// TIA Portal project "Projeto Automação Industrial" (V15.1)
// Vorlageprojekt für das Buch mit Zielsystem S7-1200

(* hardware
DEVICE "S7-1200-Station_1"  S7-1200 Station
   slot 0: "Baugruppenträger_0"  Rack  V1.0
   slot 1: "PLC_1"  CPU 1211C DC/DC/DC  6ES7 211-1AE40-0XB0  V4.1
*)

// ===== PLC "PLC_1"  CPU 1211C DC/DC/DC =====

VAR_GLOBAL   // PLC tag table "Standard-Variablentabelle"
   "Conveyor1" AT %A0.0 : Bool;
   "At exit" AT %E0.0 : Bool;
   "Start" AT %E0.1 : Bool;
   "Start light" AT %Q1.1 : Bool;
   "Start_All" AT %Q3.0 : Bool;
   "Sorter 1" AT %Q2.1 : Bool;
   "Sorter 2" AT %Q2.2 : Bool;
   "Sorter 3" AT %Q2.3 : Bool;
   "Stop blade" AT %Q0.1 : Bool;
   "Sorter 1 turn" AT %Q0.3 : Bool;
   "Sorter 1 belt" AT %Q0.4 : Bool;
   "Stop conveyor" AT %Q2.4 : Bool;
   "Vision Sensor" AT %ID30 : DInt;
   "Counter 1" AT %QD30 : DInt;
   "Stop" AT %I0.3 : Bool;
   "Counter 1 exit" AT %Q2.5 : Bool;
   "Start/stop conveyor timer" AT %Q2.6 : Bool;
   "Counter 2" AT %QD34 : DInt;
   "Counter 2 exit" AT %Q2.7 : Bool;
   "Counter 3" AT %QD38 : DInt;
   "Counter 3 exit" AT %Q1.4 : Bool;
   "Conveyor2" AT %Q0.2 : Bool;
   "Sorter 2 turn" AT %Q0.5 : Bool;
   "Sorter 2 belt" AT %Q0.6 : Bool;
   "Sorter 3 turn" AT %Q0.7 : Bool;
   "Sorter 3 belt" AT %Q1.0 : Bool;
   "Stop Light" AT %Q1.3 : Bool;
   "Exited" AT %Q3.1 : Bool;
   "Exit Timer" AT %Q3.2 : Bool;
   "Reset" AT %I0.2 : Bool;
   "Reset Light" AT %Q1.2 : Bool;
END_VAR

// folder: System blocks/Program resources

DATA_BLOCK "IEC_Counter_0_DB"   // DB1
{ S7_Optimized_Access := 'TRUE' }
AUTHOR : Simatic
FAMILY : IEC
NAME : CNTR
VERSION : 1.0
// stored: InstanceOfName IEC_COUNTER
"IEC_COUNTER"
BEGIN
END_DATA_BLOCK

DATA_BLOCK "IEC_Timer_0_DB"   // DB2
{ S7_Optimized_Access := 'TRUE' }
AUTHOR : Simatic
FAMILY : IEC
NAME : IEC_TMR
VERSION : 1.0
// stored: InstanceOfName IEC_TIMER
"IEC_TIMER"
BEGIN
END_DATA_BLOCK

DATA_BLOCK "IEC_Timer_0_DB_4"   // DB3
{ S7_Optimized_Access := 'TRUE' }
AUTHOR : Simatic
FAMILY : IEC
NAME : IEC_TMR
VERSION : 1.0
// stored: InstanceOfName IEC_TIMER
"IEC_TIMER"
BEGIN
END_DATA_BLOCK

DATA_BLOCK "IEC_Counter_0_DB_1"   // DB5
{ S7_Optimized_Access := 'TRUE' }
AUTHOR : Simatic
FAMILY : IEC
NAME : CNTR
VERSION : 1.0
// stored: InstanceOfName IEC_COUNTER
"IEC_COUNTER"
BEGIN
END_DATA_BLOCK

DATA_BLOCK "IEC_Counter_0_DB_2"   // DB6
{ S7_Optimized_Access := 'TRUE' }
AUTHOR : Simatic
FAMILY : IEC
NAME : CNTR
VERSION : 1.0
// stored: InstanceOfName IEC_COUNTER
"IEC_COUNTER"
BEGIN
END_DATA_BLOCK

DATA_BLOCK "IEC_Timer_0_DB_2"   // DB7
{ S7_Optimized_Access := 'TRUE' }
AUTHOR : Simatic
FAMILY : IEC
NAME : IEC_TMR
VERSION : 1.0
// stored: InstanceOfName IEC_TIMER
"IEC_TIMER"
BEGIN
END_DATA_BLOCK

DATA_BLOCK "IEC_Timer_0_DB_1"   // DB8
{ S7_Optimized_Access := 'TRUE' }
AUTHOR : Simatic
FAMILY : IEC
NAME : IEC_TMR
VERSION : 1.0
// stored: InstanceOfName IEC_TIMER
"IEC_TIMER"
BEGIN
END_DATA_BLOCK

DATA_BLOCK "IEC_Timer_0_DB_3"   // DB9
{ S7_Optimized_Access := 'TRUE' }
AUTHOR : Simatic
FAMILY : IEC
NAME : IEC_TMR
VERSION : 1.0
// stored: InstanceOfName IEC_TIMER
"IEC_TIMER"
BEGIN
END_DATA_BLOCK

// folder: (top level)

FUNCTION "MHJ-PLC-Lab-Function-S71200" : Void   // FC9000, SCL
{ S7_Optimized_Access := 'TRUE' }
VERSION : 0.1
   VAR_TEMP
      rdTimeReturn : Int;
      outputTime : DTL;
      SyncVal : Byte;
      forVal : Int;
      forVal_2 : Int;
      Value : Byte;
   END_VAR
   VAR CONSTANT
      CompVal : Byte := 16#34;
      Value_01 : Byte := 16#11;
      Value_01_DW : DWord := 16#A165_D992;
      Value_02_DW : DWord := 16#58BE_4401;
   END_VAR
BEGIN

   #Value:=PEEK(area := 16#82,
        dbNumber := 0,
        byteOffset := 511);
   #Value := #Value + 1;

   POKE(area := 16#82,
        dbNumber := 0,
        byteOffset := 511,
        value := #Value);

   POKE(area:=16#81,
        dbNumber:=0,
        byteOffset:=1016,
        value:=#Value_01_DW);
   POKE(area := 16#81,
        dbNumber := 0,
        byteOffset := 1020,
        value := #Value_02_DW);

   POKE(area := 16#81,
        dbNumber := 0,
        byteOffset := 511,
        value := B#16#00);

   FOR #forVal := 0 TO 120 DO
       FOR #forVal_2:=0 TO 10 DO
           #rdTimeReturn:=RD_SYS_T(#outputTime);
           #rdTimeReturn := WR_SYS_T(#outputTime);
           #rdTimeReturn := RD_SYS_T(#outputTime);
           #rdTimeReturn := WR_SYS_T(#outputTime);
       END_FOR;
       #SyncVal:= PEEK(area := 16#81,
                      dbNumber := 0,
                      byteOffset := 511);
       IF #SyncVal = #CompVal THEN
          GOTO M_1;
       END_IF;
   END_FOR;
   RETURN;

   M_1:
   POKE(area := 16#81,
        dbNumber := 0,
        byteOffset := 511,
        value := B#16#0);
END_FUNCTION

ORGANIZATION_BLOCK "Main"   // OB1, LAD, ProgramCycle
TITLE = "Main Program Sweep (Cycle)"
{ S7_Optimized_Access := 'TRUE' }
VERSION : 0.1
   VAR_INPUT
      Initial_Call : Bool;   // Initial call of this OB
      Remanence : Bool;   // =True, if remanent data are available
   END_VAR
BEGIN

REGION Network 1
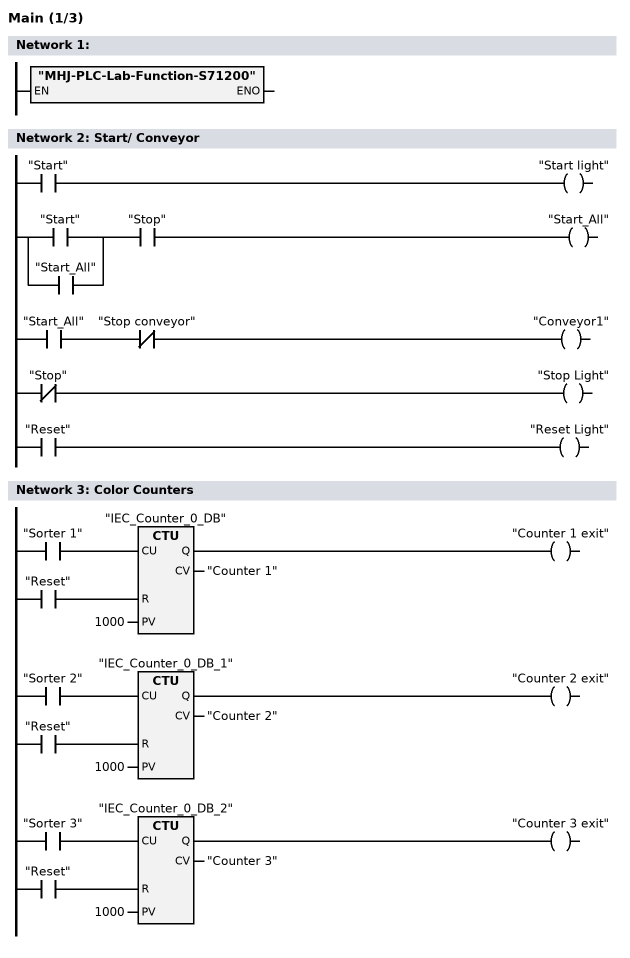
   RUNG wire#powerrail
      "MHJ-PLC-Lab-Function-S71200"()
   END_RUNG
   // the same network as SCL:
   "MHJ-PLC-Lab-Function-S71200"();
END_REGION

REGION Network 2: Start/ Conveyor
   RUNG wire#powerrail
      Contact( "Start" )
      Coil( "Start light" )
   END_RUNG
   RUNG wire#powerrail
      Contact( "Start" )
      wire#w1
      Contact( "Stop" )
      Coil( "Start_All" )
   END_RUNG
   RUNG wire#powerrail
      Contact( "Start_All" )
   END_RUNG wire#w1
   RUNG wire#powerrail
      Contact( "Start_All" )
      I_Contact( "Stop conveyor" )
      Coil( "Conveyor1" )
   END_RUNG
   RUNG wire#powerrail
      I_Contact( "Stop" )
      Coil( "Stop Light" )
   END_RUNG
   RUNG wire#powerrail
      Contact( "Reset" )
      Coil( "Reset Light" )
   END_RUNG
   // the same network as SCL:
   "Start light" := "Start";
   "Start_All" := ("Start" OR "Start_All") AND "Stop";
   "Conveyor1" := "Start_All" AND NOT "Stop conveyor";
   "Stop Light" := NOT "Stop";
   "Reset Light" := "Reset";
END_REGION

REGION Network 3: Color Counters
   "IEC_Counter_0_DB".CTU(CU := "Sorter 1", R := "Reset", PV := 1000, CV => "Counter 1");
   "Counter 1 exit" := "IEC_Counter_0_DB".Q;
   "IEC_Counter_0_DB_1".CTU(CU := "Sorter 2", R := "Reset", PV := 1000, CV => "Counter 2");
   "Counter 2 exit" := "IEC_Counter_0_DB_1".Q;
   "IEC_Counter_0_DB_2".CTU(CU := "Sorter 3", R := "Reset", PV := 1000, CV => "Counter 3");
   "Counter 3 exit" := "IEC_Counter_0_DB_2".Q;
END_REGION

REGION Network 4: Vision sensor to Sorters
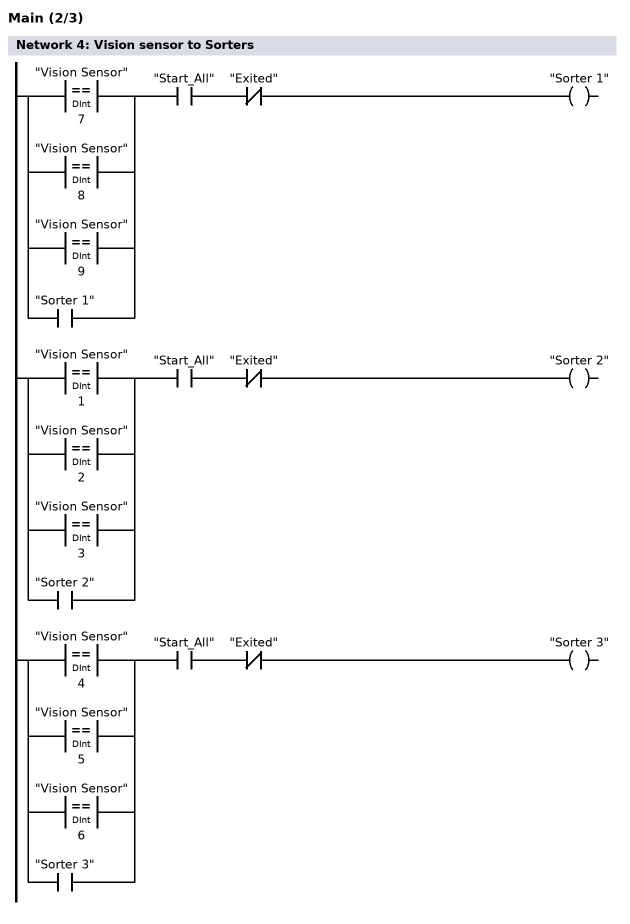
   RUNG wire#powerrail
      { S7_Templates := "SrcType := DInt" } EQ_Contact(in1 := "Vision Sensor", in2 := 7)
      wire#w1
      Contact( "Start_All" )
      I_Contact( "Exited" )
      Coil( "Sorter 1" )
   END_RUNG
   RUNG wire#powerrail
      { S7_Templates := "SrcType := DInt" } EQ_Contact(in1 := "Vision Sensor", in2 := 8)
   END_RUNG wire#w1
   RUNG wire#powerrail
      { S7_Templates := "SrcType := DInt" } EQ_Contact(in1 := "Vision Sensor", in2 := 9)
   END_RUNG wire#w1
   RUNG wire#powerrail
      Contact( "Sorter 1" )
   END_RUNG wire#w1
   RUNG wire#powerrail
      { S7_Templates := "SrcType := DInt" } EQ_Contact(in1 := "Vision Sensor", in2 := 1)
      wire#w2
      Contact( "Start_All" )
      I_Contact( "Exited" )
      Coil( "Sorter 2" )
   END_RUNG
   RUNG wire#powerrail
      { S7_Templates := "SrcType := DInt" } EQ_Contact(in1 := "Vision Sensor", in2 := 2)
   END_RUNG wire#w2
   RUNG wire#powerrail
      { S7_Templates := "SrcType := DInt" } EQ_Contact(in1 := "Vision Sensor", in2 := 3)
   END_RUNG wire#w2
   RUNG wire#powerrail
      Contact( "Sorter 2" )
   END_RUNG wire#w2
   RUNG wire#powerrail
      { S7_Templates := "SrcType := DInt" } EQ_Contact(in1 := "Vision Sensor", in2 := 4)
      wire#w3
      Contact( "Start_All" )
      I_Contact( "Exited" )
      Coil( "Sorter 3" )
   END_RUNG
   RUNG wire#powerrail
      { S7_Templates := "SrcType := DInt" } EQ_Contact(in1 := "Vision Sensor", in2 := 5)
   END_RUNG wire#w3
   RUNG wire#powerrail
      { S7_Templates := "SrcType := DInt" } EQ_Contact(in1 := "Vision Sensor", in2 := 6)
   END_RUNG wire#w3
   RUNG wire#powerrail
      Contact( "Sorter 3" )
   END_RUNG wire#w3
   // the same network as SCL:
   "Sorter 1" := (("Vision Sensor" = 7) OR ("Vision Sensor" = 8) OR ("Vision Sensor" = 9) OR "Sorter 1") AND "Start_All" AND NOT "Exited";
   "Sorter 2" := (("Vision Sensor" = 1) OR ("Vision Sensor" = 2) OR ("Vision Sensor" = 3) OR "Sorter 2") AND "Start_All" AND NOT "Exited";
   "Sorter 3" := (("Vision Sensor" = 4) OR ("Vision Sensor" = 5) OR ("Vision Sensor" = 6) OR "Sorter 3") AND "Start_All" AND NOT "Exited";
END_REGION

REGION Network 5: Turn on Sorter 1 and Sorter 2 equipment
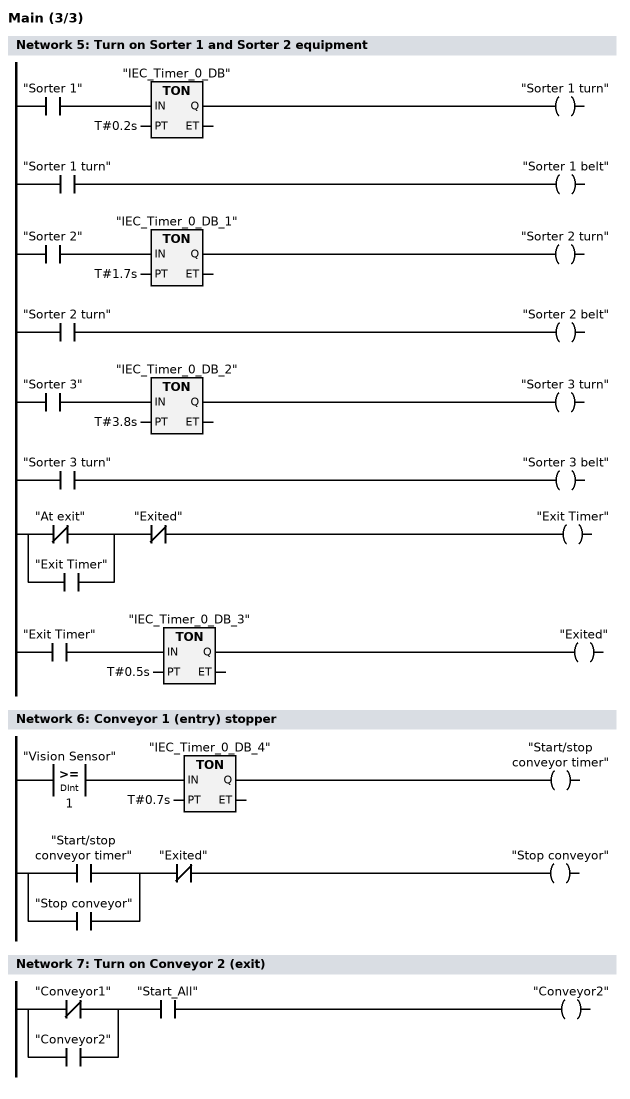
   "IEC_Timer_0_DB".TON(IN := "Sorter 1", PT := T#0.2s);
   "Sorter 1 turn" := "IEC_Timer_0_DB".Q;
   "Sorter 1 belt" := "Sorter 1 turn";
   "IEC_Timer_0_DB_1".TON(IN := "Sorter 2", PT := T#1.7s);
   "Sorter 2 turn" := "IEC_Timer_0_DB_1".Q;
   "Sorter 2 belt" := "Sorter 2 turn";
   "IEC_Timer_0_DB_2".TON(IN := "Sorter 3", PT := T#3.8s);
   "Sorter 3 turn" := "IEC_Timer_0_DB_2".Q;
   "Sorter 3 belt" := "Sorter 3 turn";
   "Exit Timer" := (NOT "At exit" OR "Exit Timer") AND NOT "Exited";
   "IEC_Timer_0_DB_3".TON(IN := "Exit Timer", PT := T#0.5s);
   "Exited" := "IEC_Timer_0_DB_3".Q;
END_REGION

REGION Network 6: Conveyor 1 (entry) stopper
   "IEC_Timer_0_DB_4".TON(IN := "Vision Sensor" >= 1, PT := T#0.7s);
   "Start/stop conveyor timer" := "IEC_Timer_0_DB_4".Q;
   "Stop conveyor" := ("Start/stop conveyor timer" OR "Stop conveyor") AND NOT "Exited";
END_REGION

REGION Network 7: Turn on Conveyor 2 (exit)
   RUNG wire#powerrail
      I_Contact( "Conveyor1" )
      wire#w1
      Contact( "Start_All" )
      Coil( "Conveyor2" )
   END_RUNG
   RUNG wire#powerrail
      Contact( "Conveyor2" )
   END_RUNG wire#w1
   // the same network as SCL:
   "Conveyor2" := (NOT "Conveyor1" OR "Conveyor2") AND "Start_All";
END_REGION
END_ORGANIZATION_BLOCK